{attribute 'linkalways'} 
{attribute 'no_explicit_call' := 'This FB is a CLASS and must be accessed using methods or properties'}
{attribute 'enable_dynamic_creation'}
FUNCTION_BLOCK FINAL NOT_BOOL EXTENDS Node
VAR
	in : _BOOL(FALSE);
	out : _BOOL(FALSE);
END_VAR

METHOD PUBLIC Clone : I_Node
VAR
	pNode : POINTER TO NOT_BOOL;
END_VAR
pNode := __NEW(NOT_BOOL);
Clone := pNode^;
END_METHOD

METHOD FB_init : BOOL
VAR_INPUT
	bInitRetains : BOOL; // if TRUE, the retain variables are initialized (warm start / cold start)
	bInCopyCode : BOOL;  // if TRUE, the instance afterwards gets moved into the copy code (online change)
END_VAR
AddInput('in',THIS^.in);
AddOutput('out', THIS^.out);
END_METHOD

METHOD PROTECTED OnExecute
VAR
END_VAR
out.Value := NOT in.Value;
END_METHOD

END_FUNCTION_BLOCK

(* stored: Version 1.1.0.1, ProductVersion 3.1.4024.15
   POU NOT_BOOL: Id {9b14e0b3-bfc8-4935-807b-c0eb53dc4784}, SpecialFunc None
   Folder Constructor: Id {98883700-f1e7-4691-bdc9-d728521fec29}
   Method Clone: Id {39e3ed62-10a8-4e0b-bfc5-c3a6098a1409}
   Method FB_init: Id {816635f4-2f6f-4665-a8ee-576f1903909b}
   Method OnExecute: Id {31465bbc-0f1e-4188-9c65-fe3ef2af70a4} *)
